{attribute 'qualified_only'}
{attribute 'strict'}
TYPE ST_RS_SeqNumber :
STRUCT
	Idle 			: BIT;
	Adsorption		: BIT;
	DeadAirEvac 	: BIT;
	SteamDesorption : BIT;
	VacCooling		: BIT;
	AirRepress 		: BIT;
	Error 			: BIT;
END_STRUCT
END_TYPE

(* stored: Version 1.1.0.1, ProductVersion 3.1.4024.12
   DUT ST_RS_SeqNumber: Id {518fea0c-aff0-4991-bbe8-8b061d65f6ed} *)
